(* PLC project Generated.project, CODESYS CODESYS V3.5 SP19 Patch 1 *)
(* stored: creationDateTime 2026-09-21T07:10:43.420112, modificationDateTime 2026-09-21T07:10:43.420112 *)

(* ═══════════════════════════════════════════════════════════════ 🎮 ST_BucketCmd — Commandes IHM pour la benne (M2) ═══════════════════════════════════════════════════════════════ *)
TYPE ST_BucketCmd : STRUCT
  BtnOpen : BOOL;  (* 🪣 Bouton commande ouverture *)
  BtnClose : BOOL;  (* 🪣 Bouton commande fermeture *)
  BtnReset : BOOL;  (* 🔑 Acquittement défaut benne *)
  BtnConfirmOpenPos : BOOL;  (* Référencement benne position ouverte (mise en service) — confirmation pure, aucun mouvement *)
  BtnConfirmClosePos : BOOL;  (* Référencement benne position fermée (mise en service) — confirmation pure, aucun mouvement *)
  BtnConfirmHomingBucket : BOOL;  (* Confirmation visuelle fermeture benne cycle homing HX1 (bouton dédié IHM) *)
  TglManualBucketLimits : BOOL := TRUE;  (* Bornes du JOG MANUEL benne -- actif uniquement en pilotage unitaire M2 (sélecteur arbitré = 2), jamais en pilotage couplé (MAINT WinchSel=0 ou SEMI_AUTO) ni pendant la phase T248. Si TRUE : borne le déplacement entre les positions ouvert/fermé configurées (OffsetOpenM/OffsetCloseM relatif à M1, mêmes bornes que FB_Bucket) ET plafonne la vitesse au palier 1, sans passer par instBucket (pas de mémorisation CloseReq/OpenReq, jogging libre borné). Défaut FALSE : jog unitaire M2 sans limite dédiée. Défaut TRUE -- jog unitaire M2 borné + palier 1 par défaut *)
  TglEnableDumpAtTremie : BOOL := FALSE;  (* Assistance "vidage à la trémie" (MAINT_N1/N2) : arme l'ouverture auto de la benne quand M3 est stable à la Trémie. Indépendant du verrou descente treuil (WinchDescentAuth_M3). *)
END_STRUCT;
END_TYPE
